(* IEC 61131-3 sources: POMIRTS_lab3/AS/Library_2/AsMc, 2 files *)

(* ---- AsMc.fun ---- *)
(********************************************************************
 * COPYRIGHT -- Bernecker + Rainer
 ********************************************************************
 * Library: AsMc
 * File: AsMc.fun
 * Author: B+R
 ********************************************************************
 * Functions and function blocks of library AsMc
 ********************************************************************)

FUNCTION MCClear : UINT		(*erases a memcard*)
END_FUNCTION

(* ---- AsMc.var ---- *)
(********************************************************************
 * COPYRIGHT -- Bernecker + Rainer
 ********************************************************************
 * Library: AsMc
 * File: AsMc.var
 * Author: B+R
 ********************************************************************
 * Local variables of library AsMc
 ********************************************************************)
VAR CONSTANT
	ERR_ASMC_ERASE_ERR	: UINT	:= 29071;		(*error erasing memcard*)
	ERR_ASMC_ERASE_OK	: UINT	:= 29070;		(*memcard erased*)
END_VAR
